Staubli VAL3: trsfDialogIns.pgx

public program trsfDialogIns(string x_sTitle, string x_sComment, trsf& x_tTrsf)
begin

  call uPage:changeTrsf(x_tTrsf, x_sTitle, x_sComment)
  call clrscr()

end
